// Block: DTrk

DATA_BLOCK DTrk
VERSION : 0.1
   NON_RETAIN
   VAR
      Empty : udt_DTrk;
      UNCUT : udt_DTrk;
      CUTTED : udt_DTrk;
      LAST_CUTTED : udt_DTrk;
   END_VAR

BEGIN
   // No initialization required
END_DATA_BLOCK
